// TwinCAT 3 PLC project PLC
// ProgramVersion: 3.1.4026.11
// libraries:
//   Tc2_Standard, * (Beckhoff Automation GmbH)
//   Tc2_System, * (Beckhoff Automation GmbH)
//   Tc2_Utilities, * (Beckhoff Automation GmbH)
//   Tc3_Module, * (Beckhoff Automation GmbH)
// project tree:
//   GVLs/ GVL.TcGVL
//   / PlcTask.TcTTO
//   POUs/ FB_Measurement.TcPOU, MAIN.TcPOU
// real-time tasks:
//   TASK PlcTask: cycle T#10ms, priority 20, ADS port 350

CONFIGURATION PLC
    RESOURCE PLC ON TwinCAT3
        TASK PlcTask(INTERVAL := T#10ms, PRIORITY := 20);
        PROGRAM MAIN WITH PlcTask : MAIN;
    END_RESOURCE
END_CONFIGURATION

// ---- GVLs/GVL.TcGVL
{attribute 'qualified_only'}
VAR_GLOBAL
	{attribute 'OPC.UA.DA' := '1'} // Enables a symbol for OPC UA.
	nMeasurement1 : LREAL;
	{attribute 'OPC.UA.DA' := '1'}
	nMeasurement2 : LREAL;
	{attribute 'OPC.UA.DA' := '1'}
	nMeasurement3 : LREAL;
	{attribute 'OPC.UA.DA' := '1'}
	nMeasurement4 : LREAL;
	{attribute 'OPC.UA.DA' := '1'}
	nMeasurement5 : LREAL;
	{attribute 'OPC.UA.DA' := '1'}
	nMeasurement6 : LREAL;
	{attribute 'OPC.UA.DA' := '1'}
	nMeasurement7 : LREAL;
	{attribute 'OPC.UA.DA' := '1'}
	nMeasurement8 : LREAL;
	{attribute 'OPC.UA.DA' := '1'}
	nMeasurement9 : LREAL;
	{attribute 'OPC.UA.DA' := '1'}
	nMeasurement10: LREAL;
	
	fbSystemTime: FB_LocalSystemTime;  // Instance of FB_LocalSystemTime
	{attribute 'OPC.UA.DA' := '1'}
    dtSystemTime: STRING;       // Variable to store the current system time
	
	{attribute 'OPC.UA.DA' := '1'}
	nMeasurement1_TimeStamp: STRING;
	{attribute 'OPC.UA.DA' := '1'}
	nMeasurement2_TimeStamp: STRING;
	{attribute 'OPC.UA.DA' := '1'}
	nMeasurement3_TimeStamp: STRING;
	{attribute 'OPC.UA.DA' := '1'}
	nMeasurement4_TimeStamp: STRING;
	{attribute 'OPC.UA.DA' := '1'}
	nMeasurement5_TimeStamp: STRING;
	{attribute 'OPC.UA.DA' := '1'}
	nMeasurement6_TimeStamp: STRING;
	{attribute 'OPC.UA.DA' := '1'}
	nMeasurement7_TimeStamp: STRING;
	{attribute 'OPC.UA.DA' := '1'}
	nMeasurement8_TimeStamp: STRING;
	{attribute 'OPC.UA.DA' := '1'}
	nMeasurement9_TimeStamp: STRING;
	{attribute 'OPC.UA.DA' := '1'}
	nMeasurement10_TimeStamp: STRING;

END_VAR

// ---- POUs/MAIN.TcPOU
PROGRAM MAIN
VAR
	fb_Measurement1: FB_Measurement;
	fb_Measurement2: FB_Measurement;
	fb_Measurement3: FB_Measurement;
END_VAR

fb_Measurement1(
	// Measurement settings
	nHighLevel:=20, 
	nLowLevel:=5 ,
	nHighDuration:=T#5S, 
	nLowDuration:=T#5S,
	nRandomizerSeedValue := 10, 
	delayTimeAfterAddOrSub :=T#100MS,
	nStepValueMult :=1,
	// Measurement value
	nMeasValue=>GVL.nMeasurement1,
	nMeasValueTimestamp => GVL.nMeasurement1_TimeStamp);
	
fb_Measurement2(
	nHighLevel:=30, 
	nLowLevel:=-30, 
	nHighDuration:=T#5S, 
	nLowDuration:=T#5S,
	nRandomizerSeedValue := 7, 
	delayTimeAfterAddOrSub :=T#100MS,
	nStepValueMult :=0.1,
	nMeasValue=>GVL.nMeasurement2,
	nMeasValueTimestamp => GVL.nMeasurement2_TimeStamp);
	
fb_Measurement3(
	nHighLevel:=-1, 
	nLowLevel:=-7, 
	nHighDuration:=T#5S, 
	nLowDuration:=T#5S,
	nRandomizerSeedValue := 42, 
	delayTimeAfterAddOrSub :=T#100MS,
	nStepValueMult :=0.01,
	nMeasValue=>GVL.nMeasurement3,
	nMeasValueTimestamp => GVL.nMeasurement3_TimeStamp);

END_PROGRAM

// ---- POUs/FB_Measurement.TcPOU
FUNCTION_BLOCK FB_Measurement
VAR_INPUT
	nHighLevel : LREAL;
	nLowLevel : REAL;
	nHighDuration : TIME;
	nLowDuration : TIME;
	nRandomizerSeedValue : INT;
	delayTimeAfterAddOrSub : TIME;
	nStepValueMult : LREAL;
END_VAR
VAR_OUTPUT
	nMeasValue : LREAL;
	nMeasValueTimestamp: STRING;
	 F_GetSystemTime   : ULINT;
END_VAR
VAR
	Randomizer : DRAND;
	TON_HighDuration : TON;
	TON_LowDuration : TON;
	TON_delayBetweenAddOrSub : TON;
	StayHighLevel : BOOL;
	StayLowLevel  : BOOL;
	is_measValueGoingUp : BOOL;
	randNum : LREAL;
    prevMeasValue: LREAL := 0.0;        // Previous measurement value

END_VAR

// initialization
TON_HighDuration.PT := nHighDuration;
TON_LowDuration.PT := nHighDuration;
Randomizer(Seed := nRandomizerSeedValue, Num => randNum);
TON_delayBetweenAddOrSub.PT := delayTimeAfterAddOrSub;

// adding delay between adding or subracting the measurement value
TON_delayBetweenAddOrSub.IN := TRUE;
IF TON_delayBetweenAddOrSub.Q THEN
	TON_delayBetweenAddOrSub.IN := FALSE;
END_IF

// Increasing measurement value
IF nMeasValue < nHighLevel AND NOT StayHighLevel AND is_measValueGoingUp THEN
	IF TON_delayBetweenAddOrSub.Q THEN
		nMeasValue := nMeasValue + nStepValueMult*randNum;
	END_IF
// Not changing measurement value when HighLevel value reached
ELSIF nMeasValue > nHighLevel AND is_measValueGoingUp THEN
	StayHighLevel := TRUE;
	TON_HighDuration.IN := TRUE;
	// Changing direction after nHighDuration
	IF TON_HighDuration.Q = TRUE THEN
		TON_HighDuration.IN := FALSE;
		StayHighLevel := FALSE;
		is_measValueGoingUp := FALSE;
	END_IF
END_IF

// Decreasing measurement value
IF nMeasValue > nLowLevel AND NOT StayLowLevel AND NOT is_measValueGoingUp THEN
	IF TON_delayBetweenAddOrSub.Q THEN
		nMeasValue := nMeasValue - nStepValueMult*randNum;
	END_IF
	
// Not changing measurement value when LowLevel value reached
ELSIF nMeasValue < nLowLevel AND NOT is_measValueGoingUp THEN
	StayLowLevel := TRUE;
	TON_LowDuration.IN := TRUE;
	// Changing direction after nLowDuration
	IF TON_LowDuration.Q = TRUE THEN
		TON_LowDuration.IN := FALSE;
		StayLowLevel := FALSE;
		is_measValueGoingUp := TRUE;
	END_IF
END_IF

// Call the FB_LocalSystemTime function block
GVL.fbSystemTime(
	sNetID:= , 
	bEnable:= TRUE, 
	dwCycle:= 1, 
	dwOpt:= , 
	tTimeout:= , 
	bValid=> , 
	systemTime=> , 
	tzID=> );
	
	GVL.dtSystemTime := SYSTEMTIME_TO_STRING(GVL.fbSystemTime.systemTime);

// Check if the measurement value has changed
IF nMeasValue <> prevMeasValue THEN
    nMeasValueTimestamp := GVL.dtSystemTime; // Update the timestamp
    prevMeasValue := nMeasValue;        // Update the previous value
END_IF

// calling timers
TON_HighDuration();
TON_LowDuration();
TON_delayBetweenAddOrSub();

END_FUNCTION_BLOCK
